TYPE ST_SafetyAliasInput :
STRUCT
	sName : STRING; //Name descriptor for the safety output
    bState : BOOL;
END_STRUCT
END_TYPE

(* stored: Version 1.1.0.1, ProductVersion 3.1.4024.11
   DUT ST_SafetyAliasInput: Id {209574b0-26ef-49a3-9c13-e6f0fed4df2d} *)
